PROGRAM Nappi_ON_OFF
VAR
	Q16: BOOL;
	Q15: BOOL;
	Q00: BOOL;
END_VAR

//P IO.in lukee napinpainalluksen nousevan aallon
//ongelmaa aikasemmin oli että kun napin laitto pohjaan niin kerran
// millisekunnissa vaihtui status
VAR // added by the converter: edge detectors and wires of the graphical bodies
    _rt1 : R_TRIG;
END_VAR

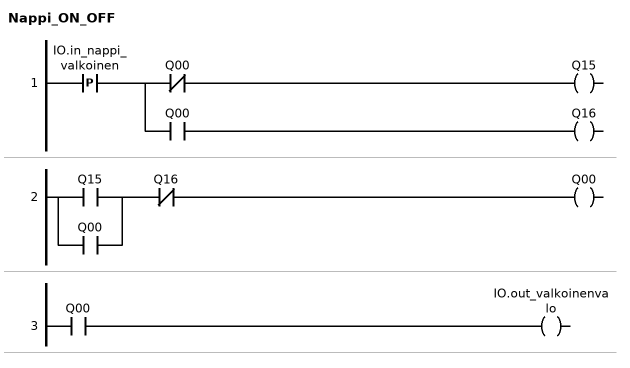
// NETWORK 1
_rt1(CLK := IO.in_nappi_valkoinen);
Q15 := _rt1.Q AND NOT Q00;
Q16 := _rt1.Q AND Q00;

// NETWORK 2
Q00 := (Q15 OR Q00) AND NOT Q16;

// NETWORK 3
IO.out_valkoinenvalo := Q00;

END_PROGRAM

(* stored: Version 1.1.0.1, ProductVersion 3.1.4024.10
   POU Nappi_ON_OFF: Id {0f98bd22-2e7d-4fd5-92db-b0eb09986945}, SpecialFunc None *)
